// TwinCAT 3 PLC project StandbyOperatingPower
// ProgramVersion: 3.1.4024.0
// libraries:
//   Tc2_Standard, * (Beckhoff Automation GmbH)
//   Tc2_System, * (Beckhoff Automation GmbH)
//   Tc3_Module, * (Beckhoff Automation GmbH)
//   VisuDialogs, * (System)
// project tree:
//   / GlobalTextList.TcGTLO, PlcTask.TcTTO, Visualization Manager.TcVMO (not stored)
//   GVLs/ GVL_IO.TcGVL
//   POUs/ FB_ToggleRelays.TcPOU, MAIN.TcPOU, ToggleRelaysWithDelay.TcPOU
//   VISUs/ Visualization.TcVIS
// real-time tasks:
//   TASK PlcTask: cycle T#10ms, priority 20, ADS port 350
// I/O:
//   DEVICE Device 5 (EtherCAT), AmsNetId 172.18.239.142.6.1
//     Term 1 (EK1100) [EK1100 EtherCAT Coupler (2A E-Bus)]
//       Term 2 (EL6070-0033) [EL6070-0033 1Ch. Licence key terminal, individual licences]
//       Term 3 (EL2809) [EL2809 16Ch. Dig. Output 24V, 0.5A]
//       Term 4 (EL2809) [EL2809 16Ch. Dig. Output 24V, 0.5A]
//       Term 5 (EL3443) [EL3443 3Ch. Power Measuring]
//       Term 6 (EL1008) [EL1008 8Ch. Dig. Input 24V, 3ms]
//       Term 7 (EL3702) [EL3702 2Ch. Ana. Input +/-10V, DIFF, Oversample]
//       Term 8 (EL9011) [EL9011 End Terminal]
//   DEVICE Device 1 (EtherCAT Automation Protocol), AmsNetId 172.18.239.142.2.1
//   DEVICE Device 2 (EtherCAT Automation Protocol), AmsNetId 172.18.239.142.3.1
//   DEVICE Device 3 (EtherCAT Automation Protocol), AmsNetId 172.18.239.142.4.1
// variable links:
//   StandbyOperatingPower/StandbyOperatingPower Instance <-> Device 5 (EtherCAT)/Term 1 (EK1100)/Term 3 (EL2809)
//     PlcTask Outputs/GVL_IO.BoolRelayArray[{1..16}] <-> Channel {1..16}/Output  (16 links)
//   StandbyOperatingPower/StandbyOperatingPower Instance <-> Device 5 (EtherCAT)/Term 1 (EK1100)/Term 4 (EL2809)
//     PlcTask Outputs/GVL_IO.BoolRelayArray[{17..22}] <-> Channel {1..6}/Output  (6 links)

CONFIGURATION StandbyOperatingPower
    RESOURCE PLC ON TwinCAT3
        TASK PlcTask(INTERVAL := T#10ms, PRIORITY := 20);
        PROGRAM MAIN WITH PlcTask : MAIN;
    END_RESOURCE
END_CONFIGURATION

// ---- GVLs/GVL_IO.TcGVL
//{attribute 'qualified_only'}   //enable this if you want to have qualified global variables, ex: GVL_IO.BoolRelayArray[]
VAR_GLOBAL
	BoolRelayArray  AT %Q* :ARRAY[1..22] OF BOOL;
	//BoolRelayArray AT %QX0.0 :ARRAY[1..21] OF BOOL;
END_VAR

// ---- POUs/MAIN.TcPOU
PROGRAM MAIN
VAR
    ToggleAllRelaysFB : FB_ToggleRelays;
    ToggleAllRelaysButton : BOOL;              // HMI toggle button
    LastToggleState: BOOL;
    ToggleRelaysWithDelayButton : BOOL;        // HMI Button
    DelayedToggle : ToggleRelaysWithDelay;     // FB Instance
    Delay : TIME;                              // TIME type, gets converted from INT
    DelayMsInput : INT;                        // User input in ms from HMI
END_VAR




// Call function block for delayed toggle
DelayedToggle(
    StartDelayToggle := ToggleRelaysWithDelayButton,
    DelayMsInput := DelayMsInput,              // Directly pass the INT to FB
    BoolRelayArray := BoolRelayArray
);

// Call function block for instant toggle
ToggleAllRelaysFB(
    ToggleButton := ToggleAllRelaysButton,
    RelayArray := BoolRelayArray
);

END_PROGRAM

// ---- POUs/FB_ToggleRelays.TcPOU
FUNCTION_BLOCK FB_ToggleRelays
VAR_INPUT
    ToggleButton: BOOL; // HMI Button
END_VAR

VAR_IN_OUT
    RelayArray : ARRAY[1..22] OF BOOL; // Global relay array
END_VAR

VAR
    LastToggleState : BOOL := FALSE;
    i : INT;
END_VAR


IF ToggleButton AND NOT LastToggleState THEN //If button is pressed, turn all relays on
    // Set all relays to OFF first
    FOR i := 1 TO 22 DO
        BoolRelayArray[i] := FALSE;
    END_FOR
	
    // Set all relays ON
    FOR i := 1 TO 22 DO
        BoolRelayArray[i] := TRUE;
    END_FOR
END_IF

// Turn all relays OFF when button returns to off state
IF NOT ToggleButton AND LastToggleState THEN  //If button gets untoggled/unpressed, turn all relays off
    FOR i := 1 TO 22 DO
        BoolRelayArray[i] := FALSE;
    END_FOR
END_IF

LastToggleState := ToggleButton; // Update the previous state of the toggle button

END_FUNCTION_BLOCK

// ---- POUs/ToggleRelaysWithDelay.TcPOU
FUNCTION_BLOCK ToggleRelaysWithDelay
VAR_INPUT
    StartDelayToggle : BOOL;           // Button from HMI
//    DelayTime : TIME := T#200MS;       // Delay between each relay
	DelayMsInput : INT; 			   // From HMI, in milliseconds
END_VAR

VAR_IN_OUT
    BoolRelayArray : ARRAY[1..22] OF BOOL; // Relay control array
END_VAR

VAR
    Timer : TON;                // Delay timer
    RelayIndex : INT := 1;      // Current relay being toggled
    Active : BOOL := FALSE;     // Whether the sequence is running
    StartLatch : BOOL := FALSE; // Edge-detection to avoid retriggering
	DelayTime : TIME; 			// Internal TIME-converted value
END_VAR


DelayTime := INT_TO_TIME(DelayMsInput);  //Convert int delay value from HIMI to type TIME

//Start the toggle sequence only once
IF StartDelayToggle AND NOT StartLatch THEN
    Active := TRUE;
    RelayIndex := 1;	//Relay index tracker
    StartLatch := TRUE;
    Timer(IN := FALSE); //Make sure timer resets
END_IF

// Reset latch when button is released
IF NOT StartDelayToggle THEN
    StartLatch := FALSE;
END_IF


// Toggle relays one-by-one with delay
IF Active THEN
    Timer(IN := TRUE, PT := DelayTime);

    IF Timer.Q THEN
        IF RelayIndex <= 22 THEN
            BoolRelayArray[RelayIndex] := TRUE;
            RelayIndex := RelayIndex + 1;	//Increment the index
            Timer(IN := FALSE); // Reset timer for next relay
        ELSE
            Active := FALSE; // Done with all relays
            Timer(IN := FALSE);
        END_IF
    END_IF
ELSE
    Timer(IN := FALSE); //Reset timer
END_IF

END_FUNCTION_BLOCK

// ---- GlobalTextList.TcGTLO
TEXTLIST GlobalTextList
  17 = '%.06'
  182 = '%.0f'
  51 = 'Control  All Relays'
  379 = 'Control All Relays'
  101 = 'Delay'
  910 = 'Delay:'
  326 = 'Individual Relay Control'
  290 = 'K1'
  882 = 'K10'
  18 = 'K11'
  621 = 'K12'
  81 = 'K13'
  772 = 'K14'
  173 = 'K15'
  721 = 'K16'
  355 = 'K17'
  258 = 'K18'
  521 = 'K19'
  193 = 'K2'
  966 = 'K20'
  813 = 'K21'
  482 = 'K22'
  839 = 'K3'
  442 = 'K4'
  132 = 'K5'
  694 = 'K6'
  914 = 'K7'
  847 = 'K8'
  480 = 'K9'
  704 = 'kk'
  974 = 'Legend'
  484 = 'LEGEND'
  683 = 'Relay 1'
  950 = 'Relay 10'
  818 = 'Relay 11'
  362 = 'Relay 12'
  126 = 'Relay 13'
  673 = 'Relay 14'
  270 = 'Relay 15'
  176 = 'Relay 16'
  183 = 'Relay 17'
  229 = 'Relay 18'
  207 = 'Relay 19'
  798 = 'Relay 2'
  38 = 'Relay 20'
  538 = 'Relay 21'
  374 = 'Relay 22'
  60 = 'Relay 3'
  392 = 'Relay 4'
  846 = 'Relay 5'
  194 = 'Relay 6'
  195 = 'Relay 7'
  235 = 'Relay 8'
  399 = 'Relay 9'
  425 = 'Relay Buttons'
  598 = 'Relay Control'
  828 = 'RELAY OFF:'
  619 = 'RELAY OFF: '
  879 = 'RELAY ON:'
  403 = 'RELAY ON: '
  600 = 'Relay Toggle Buttons'
  986 = 'RElays'
  248 = 'Relays'
  681 = 'Toggle All Relays'
  703 = 'Toggle All Relays Instantly'
  139 = 'Toggle All With Delay'
END_TEXTLIST

// ---- VISUs/Visualization.TcVIS
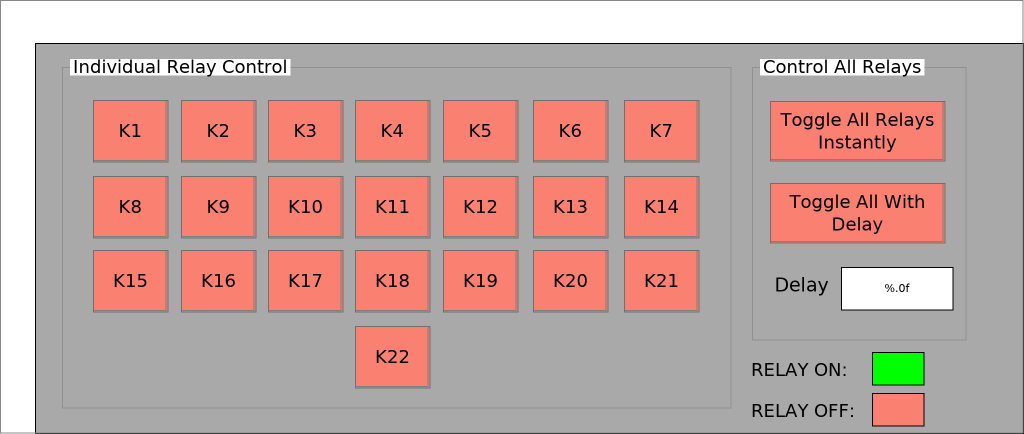
VISUALIZATION Visualization  // 1024x434
    Rectangle (35,43 989x391)
    GroupBox (62,59 669x349), "Individual Relay Control"
        Button (31,41 75x62), "K1", colour toggle: BoolRelayArray[1]
            toggle BoolRelayArray[1]
        Button (119,41 75x62), "K2", colour toggle: BoolRelayArray[2]
            toggle BoolRelayArray[2]
        Button (206,41 75x62), "K3", colour toggle: BoolRelayArray[3]
            toggle BoolRelayArray[3]
        Button (293,41 75x62), "K4", colour toggle: BoolRelayArray[4]
            toggle BoolRelayArray[4]
        Button (31,117 75x62), "K8", colour toggle: BoolRelayArray[8]
            toggle BoolRelayArray[8]
        Button (119,117 75x62), "K9", colour toggle: BoolRelayArray[9]
            toggle BoolRelayArray[9]
        Button (119,191 75x62), "K16", colour toggle: BoolRelayArray[16]
            toggle BoolRelayArray[16]
        Button (206,191 75x62), "K17", colour toggle: BoolRelayArray[17]
            toggle BoolRelayArray[17]
        Button (206,117 75x62), "K10", colour toggle: BoolRelayArray[10]
            toggle BoolRelayArray[10]
        Button (293,191 75x62), "K18", colour toggle: BoolRelayArray[18]
            toggle BoolRelayArray[18]
        Button (381,191 75x62), "K19", colour toggle: BoolRelayArray[19]
            toggle BoolRelayArray[19]
        Button (471,191 75x62), "K20", colour toggle: BoolRelayArray[20]
            toggle BoolRelayArray[20]
        Button (562,191 75x62), "K21", colour toggle: BoolRelayArray[21]
            toggle BoolRelayArray[21]
        Button (293,117 75x62), "K11", colour toggle: BoolRelayArray[11]
            toggle BoolRelayArray[11]
        Button (381,117 75x62), "K12", colour toggle: BoolRelayArray[12]
            toggle BoolRelayArray[12]
        Button (471,117 75x62), "K13", colour toggle: BoolRelayArray[13]
            toggle BoolRelayArray[13]
        Button (562,117 75x62), "K14", colour toggle: BoolRelayArray[14]
            toggle BoolRelayArray[14]
        Button (562,41 75x62), "K7", colour toggle: BoolRelayArray[7]
            toggle BoolRelayArray[7]
        Button (471,41 75x62), "K6", colour toggle: BoolRelayArray[6]
            toggle BoolRelayArray[6]
        Button (381,41 75x62), "K5", colour toggle: BoolRelayArray[5]
            toggle BoolRelayArray[5]
        Button (31,191 75x62), "K15", colour toggle: BoolRelayArray[15]
            toggle BoolRelayArray[15]
        Button (293,267 75x62), "K22", colour toggle: BoolRelayArray[21]
            toggle BoolRelayArray[22]
    GroupBox (752,59 214x281), "Control All Relays"
        Button (18,42 175x60), "Toggle All Relays Instantly", colour toggle: MAIN.ToggleRelaysWithDelayButton
            toggle MAIN.ToggleAllRelaysButton
        Button (18,124 175x60), "Toggle All With Delay", colour toggle: MAIN.ToggleRelaysWithDelayButton
            toggle MAIN.ToggleRelaysWithDelayButton
    Label (748,352 115x36), "RELAY ON:"
    Rectangle (872,352 52x33)
    Rectangle (872,393 52x33)
    Label (748,393 115x36), "RELAY OFF:"
    Label (742,270 119x30), "Delay"
    Textfield (841,267 112x43), "%.0f", text variable: MAIN.DelayMsInput
        OnMouseDown: write the text variable via Default
END_VISUALIZATION
